PROGRAM POU
VAR
	A: BOOL;
	B: BOOL;
	C: BOOL:= FALSE;
	add_result: UINT;
	sub_result: INT;
	mul_result: REAL;
	div_result: REAL;
	TON_0: TON;
	ton0_et: TIME;
	TOF_0: TOF;
	tof0_et: TIME;
	TP_0: TP;
	tp0_et: TIME;
	D: BOOL;
	CTD_0: CTD;
	CTD_1: CTD;
	ctd1_cv: WORD;
	Zero: BOOL;
	CTU_0: CTU;
	ctu0_cv: WORD;
	Maximum: BOOL;
END_VAR

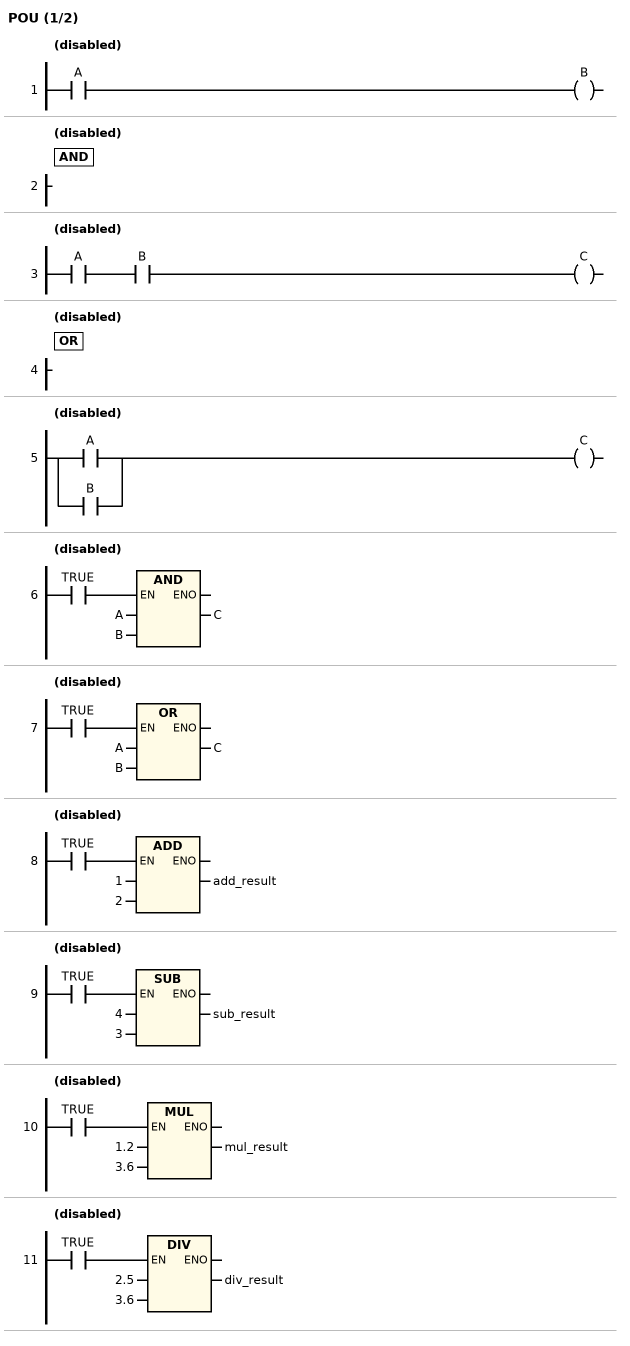
// NETWORK 1 (disabled)
// B := A;

// NETWORK 2 (disabled)
// label: AND

// NETWORK 3 (disabled)
// C := A AND B;

// NETWORK 4 (disabled)
// label: OR

// NETWORK 5 (disabled)
// C := A OR B;

// NETWORK 6 (disabled)
// C := A AND B;

// NETWORK 7 (disabled)
// C := A OR B;

// NETWORK 8 (disabled)
// add_result := 1 + 2;

// NETWORK 9 (disabled)
// sub_result := 4 - 3;

// NETWORK 10 (disabled)
// mul_result := 1.2 * 3.6;

// NETWORK 11 (disabled)
// div_result := 2.5 / 3.6;

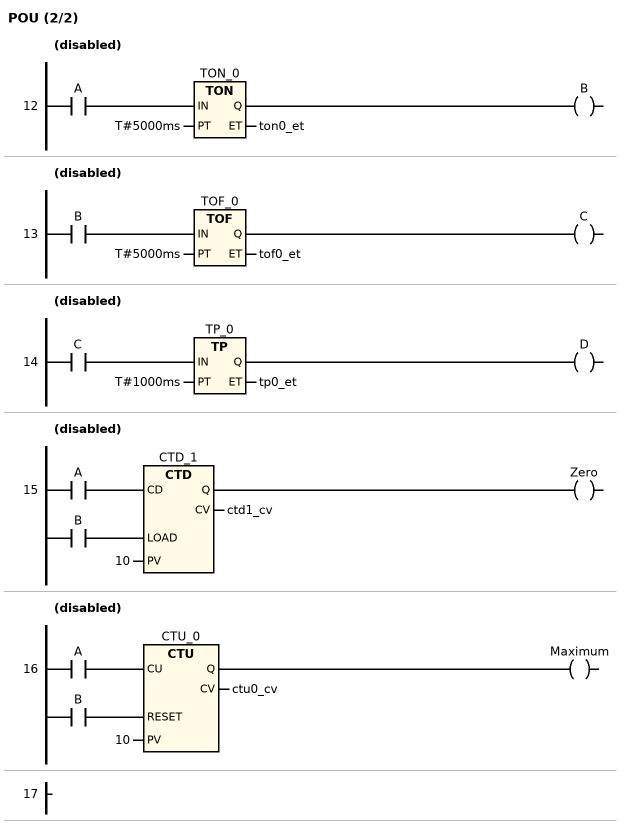
// NETWORK 12 (disabled)
// TON_0(IN := A, PT := T#5000ms, ET => ton0_et); // TON
// B := TON_0.Q;

// NETWORK 13 (disabled)
// TOF_0(IN := B, PT := T#5000ms, ET => tof0_et); // TOF
// C := TOF_0.Q;

// NETWORK 14 (disabled)
// TP_0(IN := C, PT := T#1000ms, ET => tp0_et); // TP
// D := TP_0.Q;

// NETWORK 15 (disabled)
// CTD_1(CD := A, LOAD := B, PV := 10, CV => ctd1_cv); // CTD
// Zero := CTD_1.Q;

// NETWORK 16 (disabled)
// CTU_0(CU := A, RESET := B, PV := 10, CV => ctu0_cv); // CTU
// Maximum := CTU_0.Q;

// NETWORK 17

END_PROGRAM

(* stored: Version 1.1.0.1, ProductVersion 3.1.4022.7
   POU POU: Id {b17b920c-4361-412b-ba5f-10b4e1c73886}, SpecialFunc None *)
